{attribute 'qualified_only'}
VAR_GLOBAL

END_VAR

VAR_GLOBAL CONSTANT
	MAX_DATA_LENGTH					: UINT := 32; // Data length
END_VAR

(* stored: Version 1.1.0.1, ProductVersion 3.1.4024.4
   GVL GVL_SickScanner: Id {000c2189-06cd-4623-9746-3b9af303d8b7} *)
